{attribute 'qualified_only'}
VAR_GLOBAL
	position: UINT := 0;
	velocity: UINT := 0;
	acceleration: UINT := 0;
	execute: BOOL := FALSE;
END_VAR

(* stored: Version 1.1.0.1, ProductVersion 3.1.4024.12
   GVL GVL_VARS3: Id {d280ba88-795d-4d63-830b-19e47ed8851e} *)
